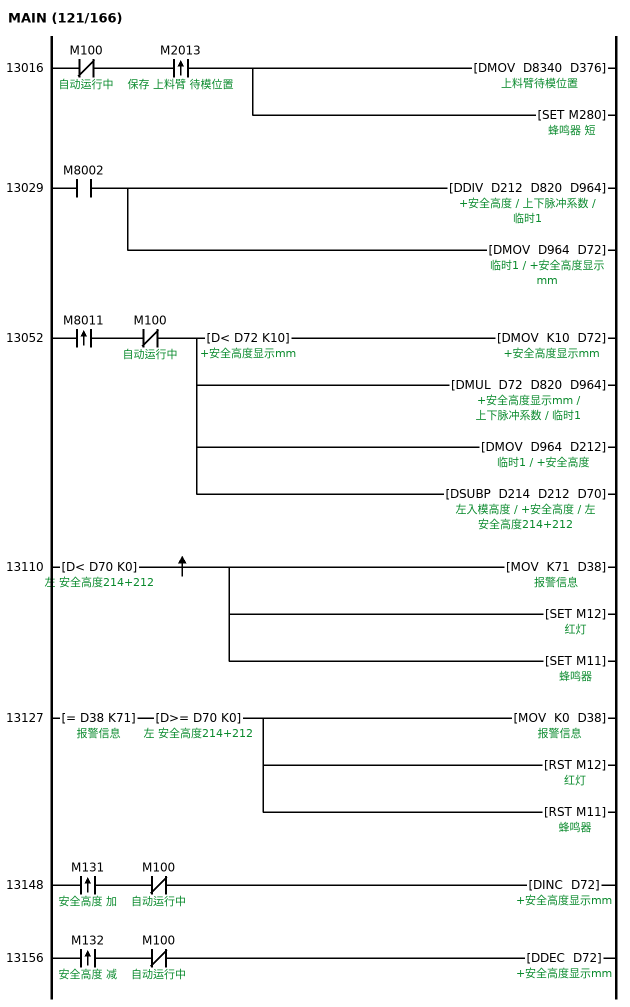
[picture p120: ladder of MAIN, rungs at steps 13016 to 13156]
13016 LDI     M100  ; 自动运行中
      ANDP    M2013  ; 保存 上料臂 待模位置
      DMOV    D8340 D376  ; 上料臂待模位置
      SET     M280  ; 蜂鸣器 短
13029 LD      M8002
      DDIV    D212 D820 D964
      DMOV    D964 D72  ; +安全高度显示mm
13052 LDP     M8011
      ANI     M100  ; 自动运行中
      MPS
      ANDD<   D72 K10  ; +安全高度显示mm
      DMOV    K10 D72
      MPP
      DMUL    D72 D820 D964
      DMOV    D964 D212
      DSUBP   D214 D212 D70
13110 LDD<    D70 K0  ; 左 安全高度214+212
      MEP
      MOV     K71 D38
      SET     M12  ; 红灯
      SET     M11  ; 蜂鸣器
13127 LD=     D38 K71  ; 报警信息
      ANDD>=  D70 K0  ; 左 安全高度214+212
      MOV     K0 D38
      RST     M12  ; 红灯
      RST     M11  ; 蜂鸣器
13148 LDP     M131  ; 安全高度 加
      ANI     M100  ; 自动运行中
      DINC    D72
13156 LDP     M132  ; 安全高度 减
      ANI     M100  ; 自动运行中
      DDEC    D72
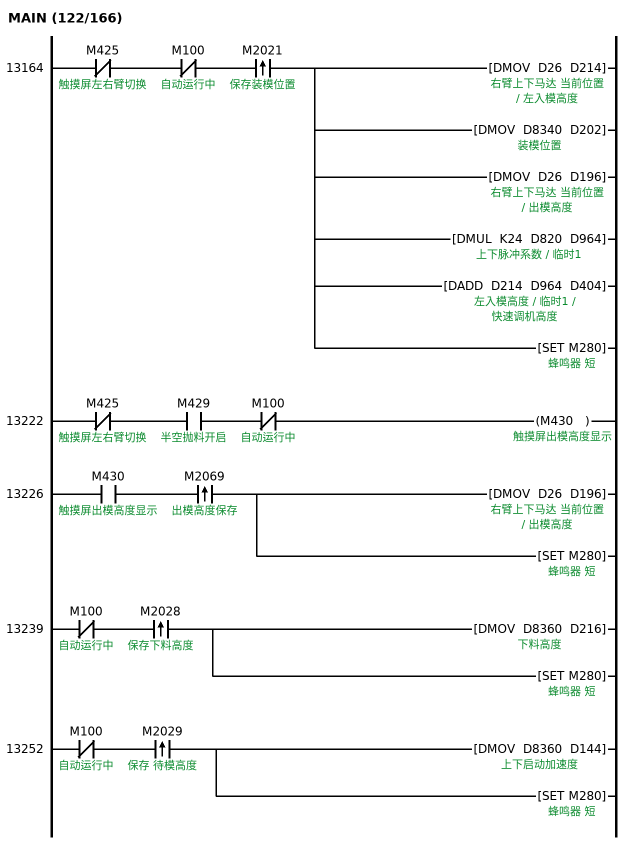
13164 LDI     M425  ; 触摸屏左右臂切换
      ANI     M100  ; 自动运行中
      ANDP    M2021  ; 保存装模位置
      DMOV    D26 D214
      DMOV    D8340 D202
      DMOV    D26 D196
      DMUL    K24 D820 D964
      DADD    D214 D964 D404
      SET     M280  ; 蜂鸣器 短
13222 LDI     M425  ; 触摸屏左右臂切换
      AND     M429  ; 半空抛料开启
      ANI     M100  ; 自动运行中
      OUT     M430  ; 触摸屏出模高度显示
13226 LD      M430  ; 触摸屏出模高度显示
      ANDP    M2069  ; 出模高度保存
      DMOV    D26 D196
      SET     M280  ; 蜂鸣器 短
13239 LDI     M100  ; 自动运行中
      ANDP    M2028  ; 保存下料高度
      DMOV    D8360 D216
      SET     M280  ; 蜂鸣器 短
13252 LDI     M100  ; 自动运行中
      ANDP    M2029  ; 保存 待模高度
      DMOV    D8360 D144  ; 上下启动加速度
      SET     M280  ; 蜂鸣器 短
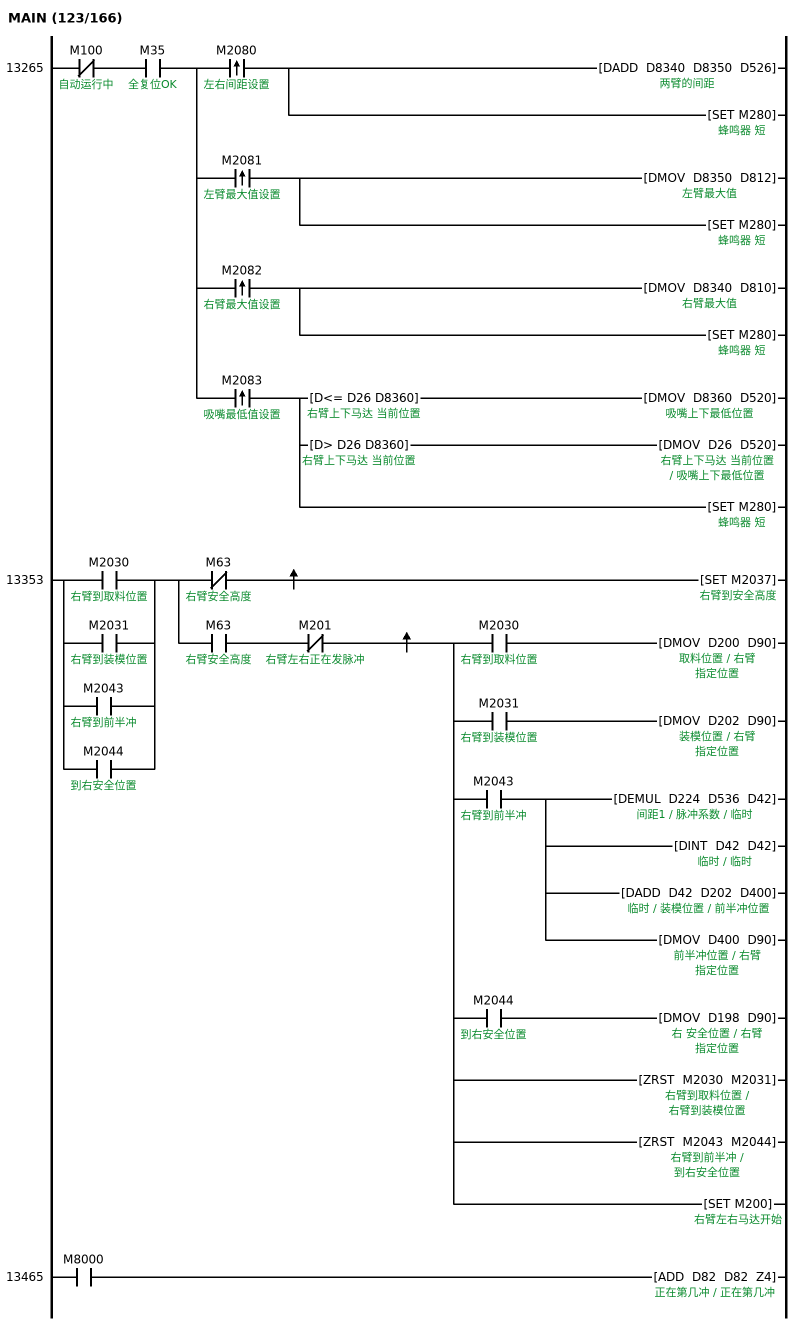
13265 LDI     M100  ; 自动运行中
      AND     M35  ; 全复位OK
      MPS
      ANDP    M2080  ; 左右间距设置
      DADD    D8340 D8350 D526
      SET     M280  ; 蜂鸣器 短
      MRD
      ANDP    M2081  ; 左臂最大值设置
      DMOV    D8350 D812
      SET     M280  ; 蜂鸣器 短
      MRD
      ANDP    M2082  ; 右臂最大值设置
      DMOV    D8340 D810
      SET     M280  ; 蜂鸣器 短
      MPP
      ANDP    M2083  ; 吸嘴最低值设置
      MPS
      ANDD<=  D26 D8360  ; 右臂上下马达 当前位置
      DMOV    D8360 D520
      MRD
      ANDD>   D26 D8360  ; 右臂上下马达 当前位置
      DMOV    D26 D520
      MPP
      SET     M280  ; 蜂鸣器 短
13353 LD      M2030  ; 右臂到取料位置
      OR      M2031  ; 右臂到装模位置
      OR      M2043  ; 右臂到前半冲
      OR      M2044  ; 到右安全位置
      MPS
      ANI     M63  ; 右臂安全高度
      MEP
      SET     M2037  ; 右臂到安全高度
      MPP
      AND     M63  ; 右臂安全高度
      ANI     M201  ; 右臂左右正在发脉冲
      MEP
      MPS
      AND     M2030  ; 右臂到取料位置
      DMOV    D200 D90
      MRD
      AND     M2031  ; 右臂到装模位置
      DMOV    D202 D90
      MRD
      AND     M2043  ; 右臂到前半冲
      DEMUL   D224 D536 D42
      DINT    D42 D42
      DADD    D42 D202 D400
      DMOV    D400 D90
      MRD
      AND     M2044  ; 到右安全位置
      DMOV    D198 D90
      MPP
      ZRST    M2030 M2031
      ZRST    M2043 M2044
      SET     M200  ; 右臂左右马达开始
13465 LD      M8000
      ADD     D82 D82 Z4
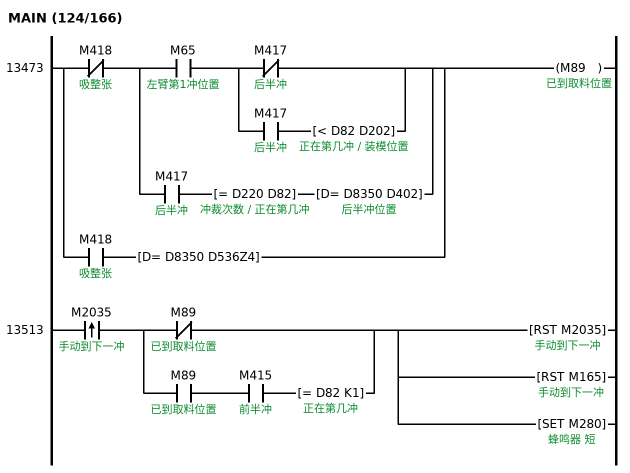
13473 LDI     M418  ; 吸整张
      LD      M65  ; 左臂第1冲位置
      LDI     M417  ; 后半冲
      LD      M417  ; 后半冲
      AND<    D82 D202  ; 正在第几冲 / 装模位置
      ORB
      ANB
      LD      M417  ; 后半冲
      AND=    D220 D82  ; 冲裁次数 / 正在第几冲
      ANDD=   D8350 D402  ; 后半冲位置
      ORB
      ANB
      LD      M418  ; 吸整张
      ANDD=   D8350 D536Z4
      ORB
      OUT     M89  ; 已到取料位置
13513 LDP     M2035  ; 手动到下一冲
      LDI     M89  ; 已到取料位置
      LD      M89  ; 已到取料位置
      AND     M415  ; 前半冲
      AND=    D82 K1  ; 正在第几冲
      ORB
      ANB
      RST     M2035  ; 手动到下一冲
      RST     M165  ; 手动到下一冲
      SET     M280  ; 蜂鸣器 短
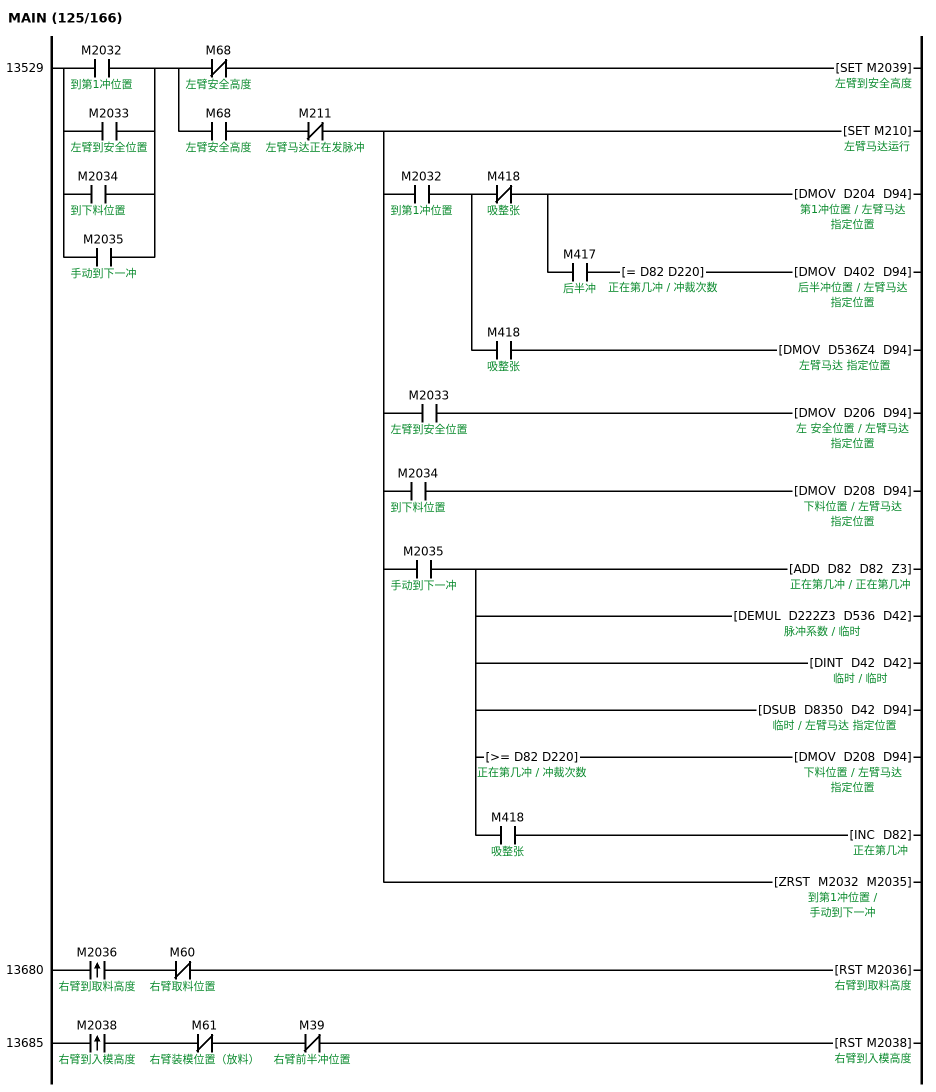
13529 LD      M2032  ; 到第1冲位置
      OR      M2033  ; 左臂到安全位置
      OR      M2034  ; 到下料位置
      OR      M2035  ; 手动到下一冲
      MPS
      ANI     M68  ; 左臂安全高度
      SET     M2039  ; 左臂到安全高度
      MPP
      AND     M68  ; 左臂安全高度
      ANI     M211  ; 左臂马达正在发脉冲
      SET     M210  ; 左臂马达运行
      MPS
      AND     M2032  ; 到第1冲位置
      MPS
      ANI     M418  ; 吸整张
      DMOV    D204 D94
      AND     M417  ; 后半冲
      AND=    D82 D220  ; 正在第几冲 / 冲裁次数
      DMOV    D402 D94
      MPP
      AND     M418  ; 吸整张
      DMOV    D536Z4 D94
      MRD
      AND     M2033  ; 左臂到安全位置
      DMOV    D206 D94
      MRD
      AND     M2034  ; 到下料位置
      DMOV    D208 D94
      MRD
      AND     M2035  ; 手动到下一冲
      ADD     D82 D82 Z3
      DEMUL   D222Z3 D536 D42
      DINT    D42 D42
      DSUB    D8350 D42 D94
      MPS
      AND>=   D82 D220  ; 正在第几冲 / 冲裁次数
      DMOV    D208 D94
      MPP
      AND     M418  ; 吸整张
      INC     D82
      MPP
      ZRST    M2032 M2035
13680 LDP     M2036  ; 右臂到取料高度
      ANI     M60  ; 右臂取料位置
      RST     M2036  ; 右臂到取料高度
13685 LDP     M2038  ; 右臂到入模高度
      ANI     M61  ; 右臂装模位置（放料）
      ANI     M39  ; 右臂前半冲位置
      RST     M2038  ; 右臂到入模高度
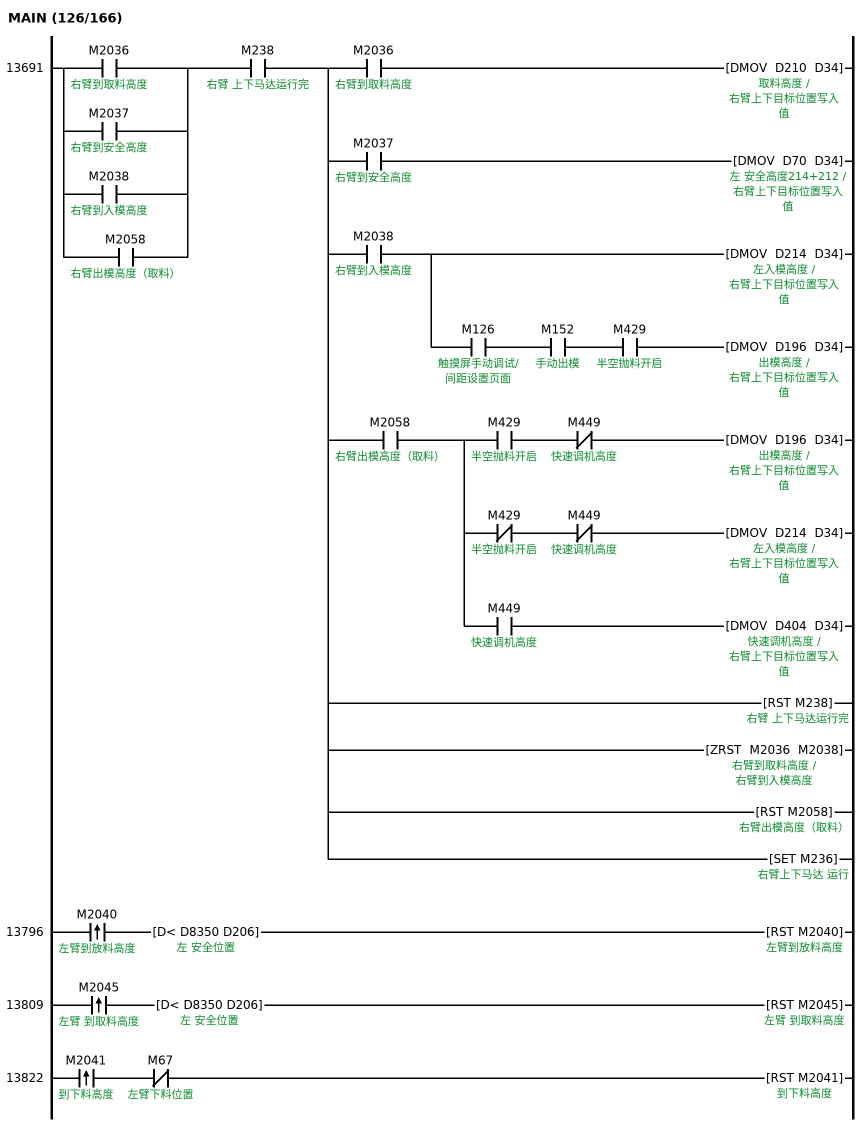
13691 LD      M2036  ; 右臂到取料高度
      OR      M2037  ; 右臂到安全高度
      OR      M2038  ; 右臂到入模高度
      OR      M2058  ; 右臂出模高度（取料）
      AND     M238  ; 右臂 上下马达运行完
      MPS
      AND     M2036  ; 右臂到取料高度
      DMOV    D210 D34
      MRD
      AND     M2037  ; 右臂到安全高度
      DMOV    D70 D34
      MRD
      AND     M2038  ; 右臂到入模高度
      DMOV    D214 D34
      AND     M126  ; 触摸屏手动调试/间距设置页面
      AND     M152  ; 手动出模
      AND     M429  ; 半空抛料开启
      DMOV    D196 D34
      MRD
      AND     M2058  ; 右臂出模高度（取料）
      MPS
      AND     M429  ; 半空抛料开启
      ANI     M449  ; 快速调机高度
      DMOV    D196 D34
      MRD
      ANI     M429  ; 半空抛料开启
      ANI     M449  ; 快速调机高度
      DMOV    D214 D34
      MPP
      AND     M449  ; 快速调机高度
      DMOV    D404 D34
      MPP
      RST     M238  ; 右臂 上下马达运行完
      ZRST    M2036 M2038
      RST     M2058  ; 右臂出模高度（取料）
      SET     M236  ; 右臂上下马达 运行
13796 LDP     M2040  ; 左臂到放料高度
      ANDD<   D8350 D206  ; 左 安全位置
      RST     M2040  ; 左臂到放料高度
13809 LDP     M2045  ; 左臂 到取料高度
      ANDD<   D8350 D206  ; 左 安全位置
      RST     M2045  ; 左臂 到取料高度
13822 LDP     M2041  ; 到下料高度
      ANI     M67  ; 左臂下料位置
      RST     M2041  ; 到下料高度
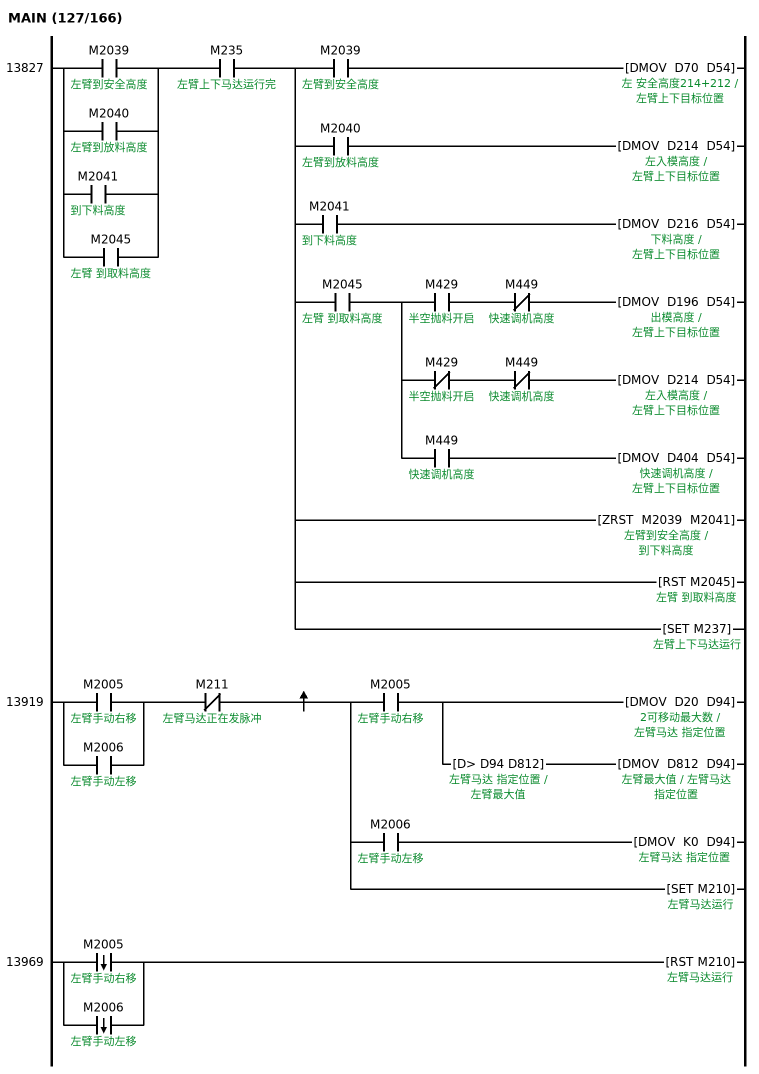
13827 LD      M2039  ; 左臂到安全高度
      OR      M2040  ; 左臂到放料高度
      OR      M2041  ; 到下料高度
      OR      M2045  ; 左臂 到取料高度
      AND     M235  ; 左臂上下马达运行完
      MPS
      AND     M2039  ; 左臂到安全高度
      DMOV    D70 D54
      MRD
      AND     M2040  ; 左臂到放料高度
      DMOV    D214 D54
      MRD
      AND     M2041  ; 到下料高度
      DMOV    D216 D54
      MRD
      AND     M2045  ; 左臂 到取料高度
      MPS
      AND     M429  ; 半空抛料开启
      ANI     M449  ; 快速调机高度
      DMOV    D196 D54
      MRD
      ANI     M429  ; 半空抛料开启
      ANI     M449  ; 快速调机高度
      DMOV    D214 D54
      MPP
      AND     M449  ; 快速调机高度
      DMOV    D404 D54
      MPP
      ZRST    M2039 M2041
      RST     M2045  ; 左臂 到取料高度
      SET     M237  ; 左臂上下马达运行
13919 LD      M2005  ; 左臂手动右移
      OR      M2006  ; 左臂手动左移
      ANI     M211  ; 左臂马达正在发脉冲
      MEP
      MPS
      AND     M2005  ; 左臂手动右移
      DMOV    D20 D94
      ANDD>   D94 D812  ; 左臂马达 指定位置 / 左臂最大值
      DMOV    D812 D94
      MRD
      AND     M2006  ; 左臂手动左移
      DMOV    K0 D94
      MPP
      SET     M210  ; 左臂马达运行
13969 LDF     M2005  ; 左臂手动右移
      ORF     M2006  ; 左臂手动左移
      RST     M210  ; 左臂马达运行
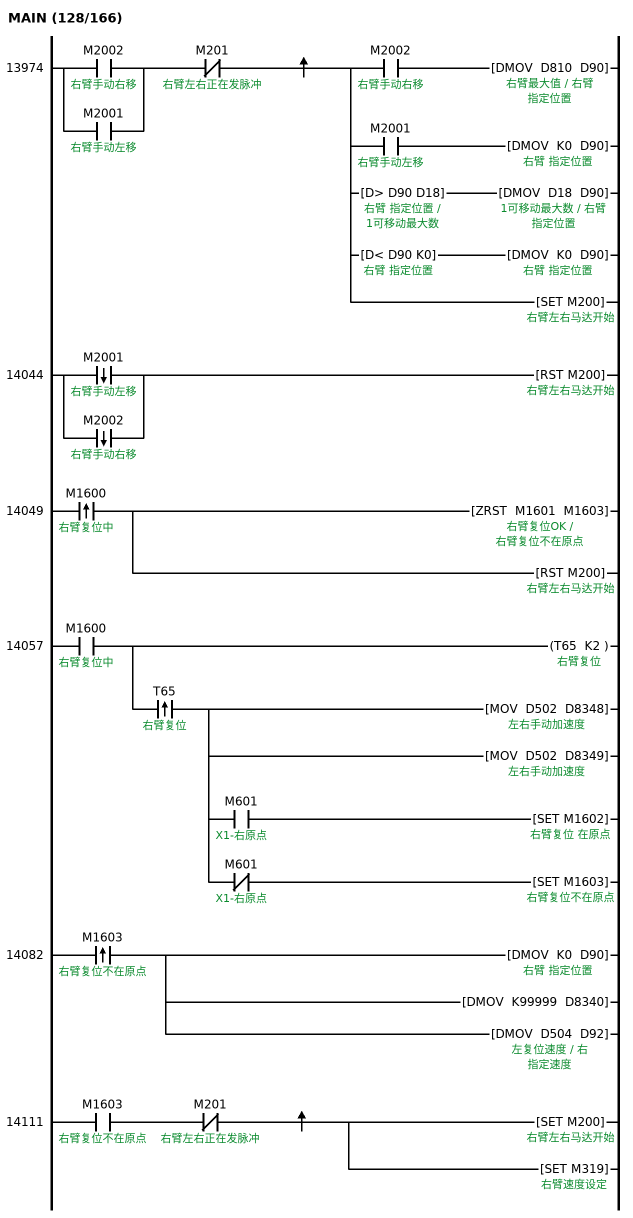
13974 LD      M2002  ; 右臂手动右移
      OR      M2001  ; 右臂手动左移
      ANI     M201  ; 右臂左右正在发脉冲
      MEP
      MPS
      AND     M2002  ; 右臂手动右移
      DMOV    D810 D90
      MRD
      AND     M2001  ; 右臂手动左移
      DMOV    K0 D90
      MRD
      ANDD>   D90 D18  ; 右臂 指定位置 / 1可移动最大数
      DMOV    D18 D90
      MRD
      ANDD<   D90 K0  ; 右臂 指定位置
      DMOV    K0 D90
      MPP
      SET     M200  ; 右臂左右马达开始
14044 LDF     M2001  ; 右臂手动左移
      ORF     M2002  ; 右臂手动右移
      RST     M200  ; 右臂左右马达开始
14049 LDP     M1600  ; 右臂复位中
      ZRST    M1601 M1603  ; 右臂复位不在原点
      RST     M200  ; 右臂左右马达开始
14057 LD      M1600  ; 右臂复位中
      OUT     T65 K2  ; 右臂复位
      ANDP    T65  ; 右臂复位
      MOV     D502 D8348
      MOV     D502 D8349
      MPS
      AND     M601  ; X1-右原点
      SET     M1602  ; 右臂复位 在原点
      MPP
      ANI     M601  ; X1-右原点
      SET     M1603  ; 右臂复位不在原点
14082 LDP     M1603  ; 右臂复位不在原点
      DMOV    K0 D90
      DMOV    K99999 D8340
      DMOV    D504 D92  ; 右 指定速度
14111 LD      M1603  ; 右臂复位不在原点
      ANI     M201  ; 右臂左右正在发脉冲
      MEP
      SET     M200  ; 右臂左右马达开始
      SET     M319  ; 右臂速度设定
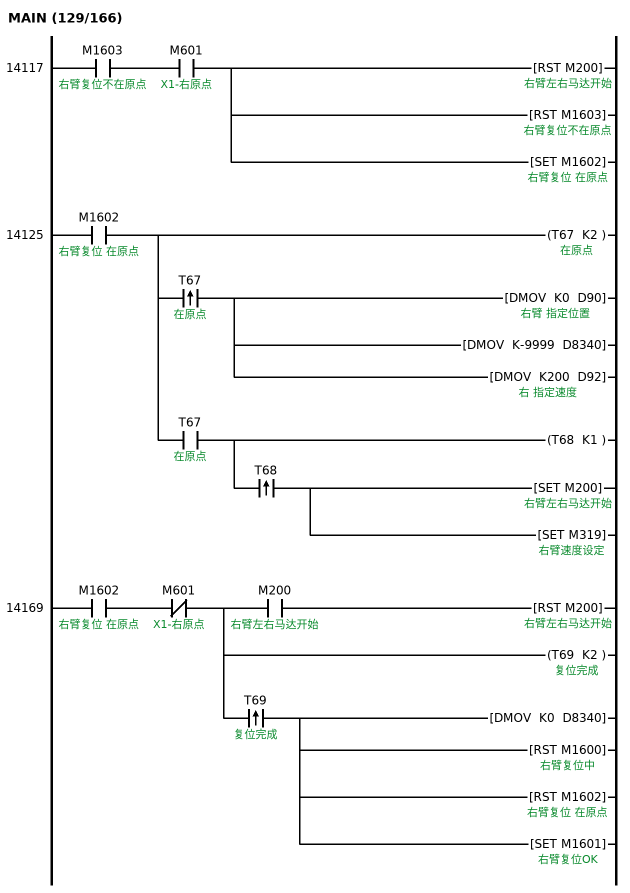
14117 LD      M1603  ; 右臂复位不在原点
      AND     M601  ; X1-右原点
      RST     M200  ; 右臂左右马达开始
      RST     M1603  ; 右臂复位不在原点
      SET     M1602  ; 右臂复位 在原点
14125 LD      M1602  ; 右臂复位 在原点
      OUT     T67 K2  ; 在原点
      MPS
      ANDP    T67  ; 在原点
      DMOV    K0 D90
      DMOV    K-9999 D8340
      DMOV    K200 D92
      MPP
      AND     T67  ; 在原点
      OUT     T68 K1
      ANDP    T68
      SET     M200  ; 右臂左右马达开始
      SET     M319  ; 右臂速度设定
14169 LD      M1602  ; 右臂复位 在原点
      ANI     M601  ; X1-右原点
      MPS
      AND     M200  ; 右臂左右马达开始
      RST     M200  ; 右臂左右马达开始
      MPP
      OUT     T69 K2  ; 复位完成
      ANDP    T69  ; 复位完成
      DMOV    K0 D8340
      RST     M1600  ; 右臂复位中
      RST     M1602  ; 右臂复位 在原点
      SET     M1601  ; 右臂复位OK
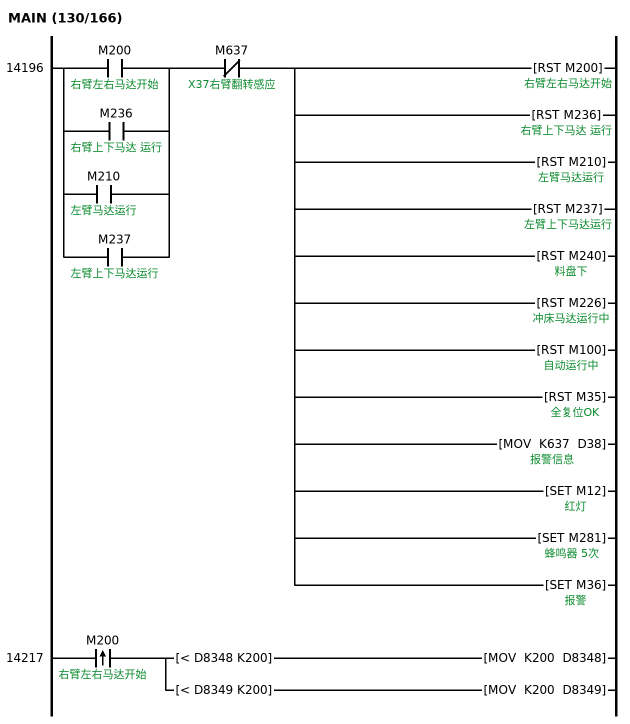
14196 LD      M200  ; 右臂左右马达开始
      OR      M236  ; 右臂上下马达 运行
      OR      M210  ; 左臂马达运行
      OR      M237  ; 左臂上下马达运行
      ANI     M637  ; X37右臂翻转感应
      RST     M200  ; 右臂左右马达开始
      RST     M236  ; 右臂上下马达 运行
      RST     M210  ; 左臂马达运行
      RST     M237  ; 左臂上下马达运行
      RST     M240  ; 料盘下
      RST     M226  ; 冲床马达运行中
      RST     M100  ; 自动运行中
      RST     M35  ; 全复位OK
      MOV     K637 D38
      SET     M12  ; 红灯
      SET     M281  ; 蜂鸣器 5次
      SET     M36  ; 报警
14217 LDP     M200  ; 右臂左右马达开始
      MPS
      AND<    D8348 K200
      MOV     K200 D8348
      MPP
      AND<    D8349 K200
      MOV     K200 D8349
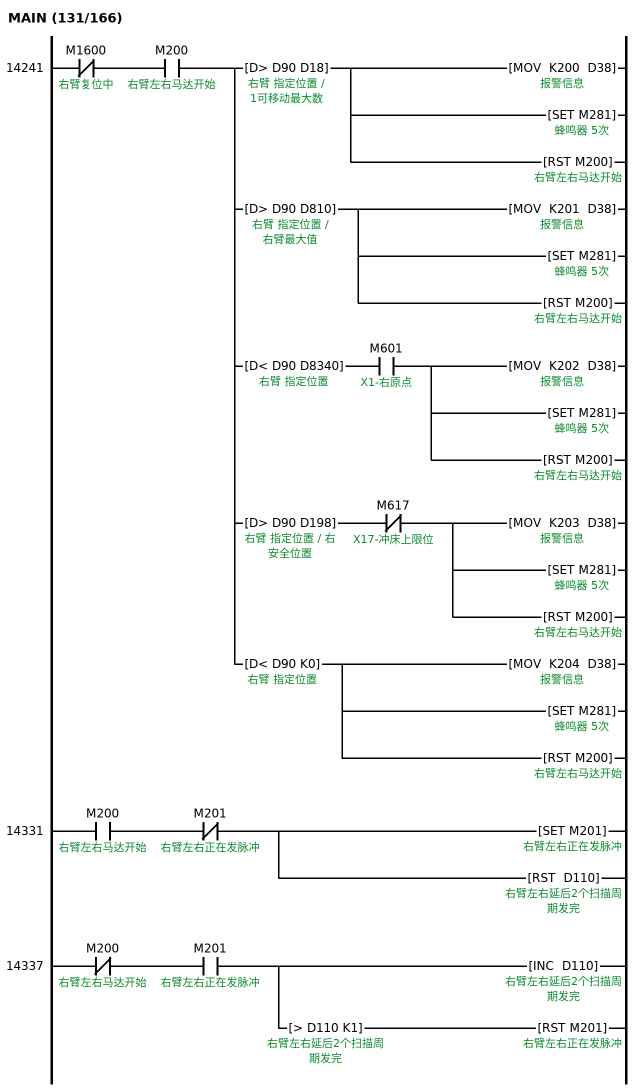
14241 LDI     M1600  ; 右臂复位中
      AND     M200  ; 右臂左右马达开始
      MPS
      ANDD>   D90 D18  ; 右臂 指定位置 / 1可移动最大数
      MOV     K200 D38
      SET     M281  ; 蜂鸣器 5次
      RST     M200  ; 右臂左右马达开始
      MRD
      ANDD>   D90 D810  ; 右臂 指定位置 / 右臂最大值
      MOV     K201 D38
      SET     M281  ; 蜂鸣器 5次
      RST     M200  ; 右臂左右马达开始
      MRD
      ANDD<   D90 D8340  ; 右臂 指定位置
      AND     M601  ; X1-右原点
      MOV     K202 D38
      SET     M281  ; 蜂鸣器 5次
      RST     M200  ; 右臂左右马达开始
      MRD
      ANDD>   D90 D198  ; 右臂 指定位置 / 右 安全位置
      ANI     M617  ; X17-冲床上限位
      MOV     K203 D38
      SET     M281  ; 蜂鸣器 5次
      RST     M200  ; 右臂左右马达开始
      MPP
      ANDD<   D90 K0  ; 右臂 指定位置
      MOV     K204 D38
      SET     M281  ; 蜂鸣器 5次
      RST     M200  ; 右臂左右马达开始
14331 LD      M200  ; 右臂左右马达开始
      ANI     M201  ; 右臂左右正在发脉冲
      SET     M201  ; 右臂左右正在发脉冲
      RST     D110  ; 右臂左右延后2个扫描周期发完
14337 LDI     M200  ; 右臂左右马达开始
      AND     M201  ; 右臂左右正在发脉冲
      INC     D110
      AND>    D110 K1  ; 右臂左右延后2个扫描周期发完
      RST     M201  ; 右臂左右正在发脉冲
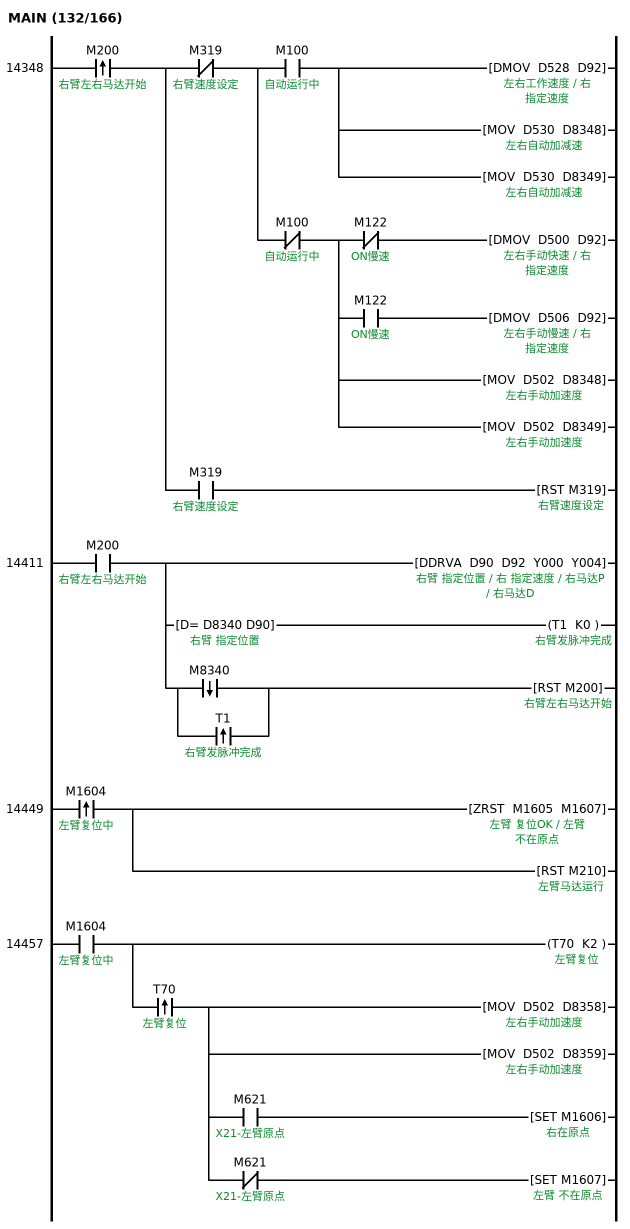
14348 LDP     M200  ; 右臂左右马达开始
      MPS
      ANI     M319  ; 右臂速度设定
      MPS
      AND     M100  ; 自动运行中
      DMOV    D528 D92
      MOV     D530 D8348
      MOV     D530 D8349
      MPP
      ANI     M100  ; 自动运行中
      MPS
      ANI     M122  ; ON慢速
      DMOV    D500 D92
      MRD
      AND     M122  ; ON慢速
      DMOV    D506 D92
      MPP
      MOV     D502 D8348
      MOV     D502 D8349
      MPP
      AND     M319  ; 右臂速度设定
      RST     M319  ; 右臂速度设定
14411 LD      M200  ; 右臂左右马达开始
      DDRVA   D90 D92 Y000 Y004  ; 右马达P / 右马达D
      MPS
      ANDD=   D8340 D90  ; 右臂 指定位置
      OUT     T1 K0  ; 右臂发脉冲完成
      MPP
      LDF     M8340
      ORP     T1  ; 右臂发脉冲完成
      ANB
      RST     M200  ; 右臂左右马达开始
14449 LDP     M1604  ; 左臂复位中
      ZRST    M1605 M1607  ; 左臂 不在原点
      RST     M210  ; 左臂马达运行
14457 LD      M1604  ; 左臂复位中
      OUT     T70 K2  ; 左臂复位
      ANDP    T70  ; 左臂复位
      MOV     D502 D8358
      MOV     D502 D8359
      MPS
      AND     M621  ; X21-左臂原点
      SET     M1606  ; 右在原点
      MPP
      ANI     M621  ; X21-左臂原点
      SET     M1607  ; 左臂 不在原点
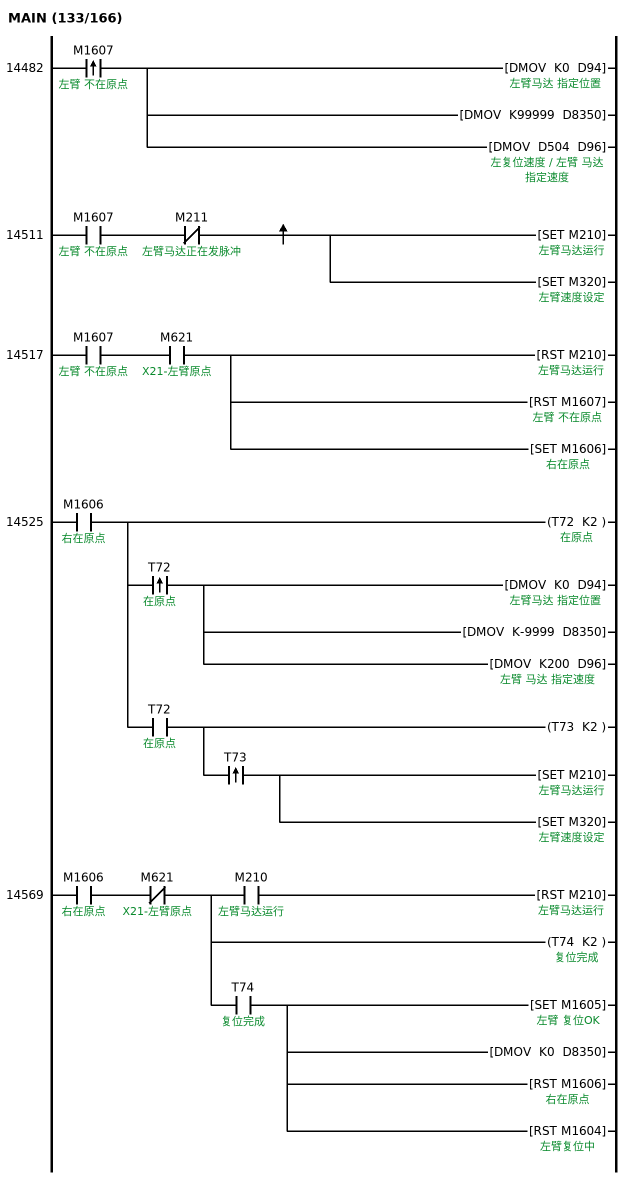
14482 LDP     M1607  ; 左臂 不在原点
      DMOV    K0 D94
      DMOV    K99999 D8350
      DMOV    D504 D96  ; 左臂 马达 指定速度
14511 LD      M1607  ; 左臂 不在原点
      ANI     M211  ; 左臂马达正在发脉冲
      MEP
      SET     M210  ; 左臂马达运行
      SET     M320  ; 左臂速度设定
14517 LD      M1607  ; 左臂 不在原点
      AND     M621  ; X21-左臂原点
      RST     M210  ; 左臂马达运行
      RST     M1607  ; 左臂 不在原点
      SET     M1606  ; 右在原点
14525 LD      M1606  ; 右在原点
      OUT     T72 K2  ; 在原点
      MPS
      ANDP    T72  ; 在原点
      DMOV    K0 D94
      DMOV    K-9999 D8350
      DMOV    K200 D96
      MPP
      AND     T72  ; 在原点
      OUT     T73 K2
      ANDP    T73
      SET     M210  ; 左臂马达运行
      SET     M320  ; 左臂速度设定
14569 LD      M1606  ; 右在原点
      ANI     M621  ; X21-左臂原点
      MPS
      AND     M210  ; 左臂马达运行
      RST     M210  ; 左臂马达运行
      MPP
      OUT     T74 K2  ; 复位完成
      AND     T74  ; 复位完成
      SET     M1605  ; 左臂 复位OK
      DMOV    K0 D8350
      RST     M1606  ; 右在原点
      RST     M1604  ; 左臂复位中
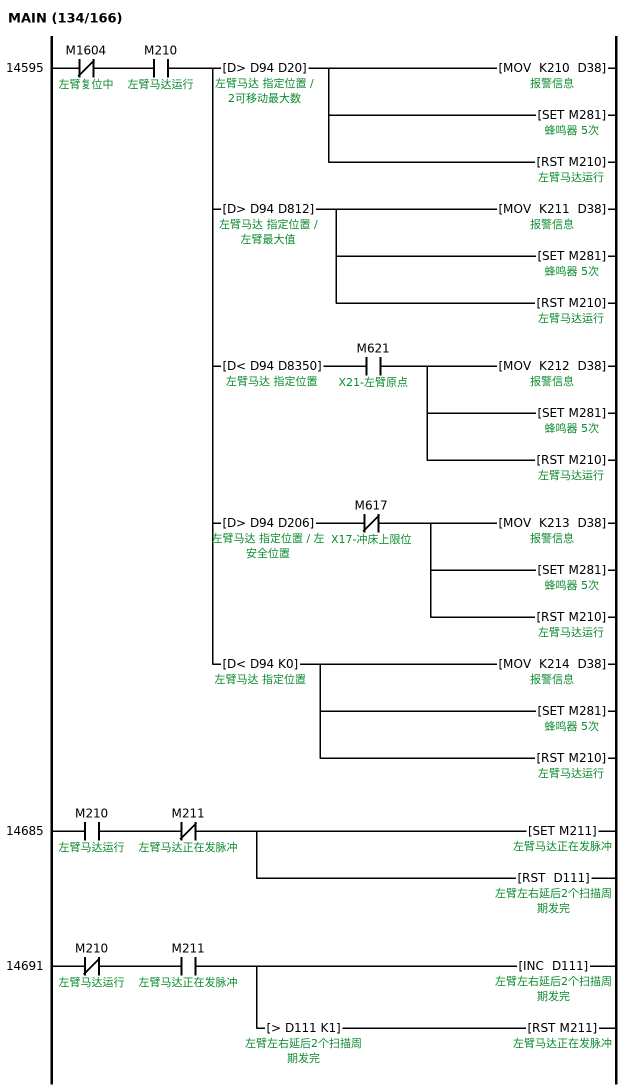
14595 LDI     M1604  ; 左臂复位中
      AND     M210  ; 左臂马达运行
      MPS
      ANDD>   D94 D20  ; 左臂马达 指定位置 / 2可移动最大数
      MOV     K210 D38
      SET     M281  ; 蜂鸣器 5次
      RST     M210  ; 左臂马达运行
      MRD
      ANDD>   D94 D812  ; 左臂马达 指定位置 / 左臂最大值
      MOV     K211 D38
      SET     M281  ; 蜂鸣器 5次
      RST     M210  ; 左臂马达运行
      MRD
      ANDD<   D94 D8350  ; 左臂马达 指定位置
      AND     M621  ; X21-左臂原点
      MOV     K212 D38
      SET     M281  ; 蜂鸣器 5次
      RST     M210  ; 左臂马达运行
      MRD
      ANDD>   D94 D206  ; 左臂马达 指定位置 / 左 安全位置
      ANI     M617  ; X17-冲床上限位
      MOV     K213 D38
      SET     M281  ; 蜂鸣器 5次
      RST     M210  ; 左臂马达运行
      MPP
      ANDD<   D94 K0  ; 左臂马达 指定位置
      MOV     K214 D38
      SET     M281  ; 蜂鸣器 5次
      RST     M210  ; 左臂马达运行
14685 LD      M210  ; 左臂马达运行
      ANI     M211  ; 左臂马达正在发脉冲
      SET     M211  ; 左臂马达正在发脉冲
      RST     D111  ; 左臂左右延后2个扫描周期发完
14691 LDI     M210  ; 左臂马达运行
      AND     M211  ; 左臂马达正在发脉冲
      INC     D111
      AND>    D111 K1  ; 左臂左右延后2个扫描周期发完
      RST     M211  ; 左臂马达正在发脉冲
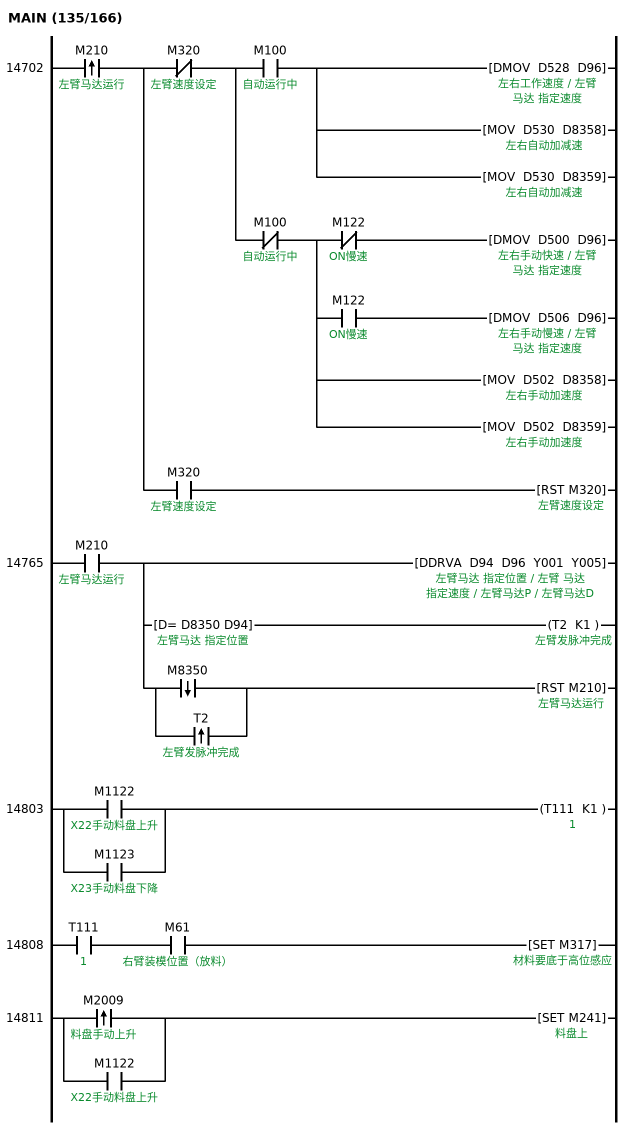
14702 LDP     M210  ; 左臂马达运行
      MPS
      ANI     M320  ; 左臂速度设定
      MPS
      AND     M100  ; 自动运行中
      DMOV    D528 D96
      MOV     D530 D8358
      MOV     D530 D8359
      MPP
      ANI     M100  ; 自动运行中
      MPS
      ANI     M122  ; ON慢速
      DMOV    D500 D96
      MRD
      AND     M122  ; ON慢速
      DMOV    D506 D96
      MPP
      MOV     D502 D8358
      MOV     D502 D8359
      MPP
      AND     M320  ; 左臂速度设定
      RST     M320  ; 左臂速度设定
14765 LD      M210  ; 左臂马达运行
      DDRVA   D94 D96 Y001 Y005  ; 左臂马达P / 左臂马达D
      MPS
      ANDD=   D8350 D94  ; 左臂马达 指定位置
      OUT     T2 K1  ; 左臂发脉冲完成
      MPP
      LDF     M8350
      ORP     T2  ; 左臂发脉冲完成
      ANB
      RST     M210  ; 左臂马达运行
14803 LD      M1122  ; X22手动料盘上升
      OR      M1123  ; X23手动料盘下降
      OUT     T111 K1  ; 1
14808 LD      T111  ; 1
      AND     M61  ; 右臂装模位置（放料）
      SET     M317  ; 材料要底于高位感应
14811 LDP     M2009  ; 料盘手动上升
      OR      M1122  ; X22手动料盘上升
      SET     M241  ; 料盘上
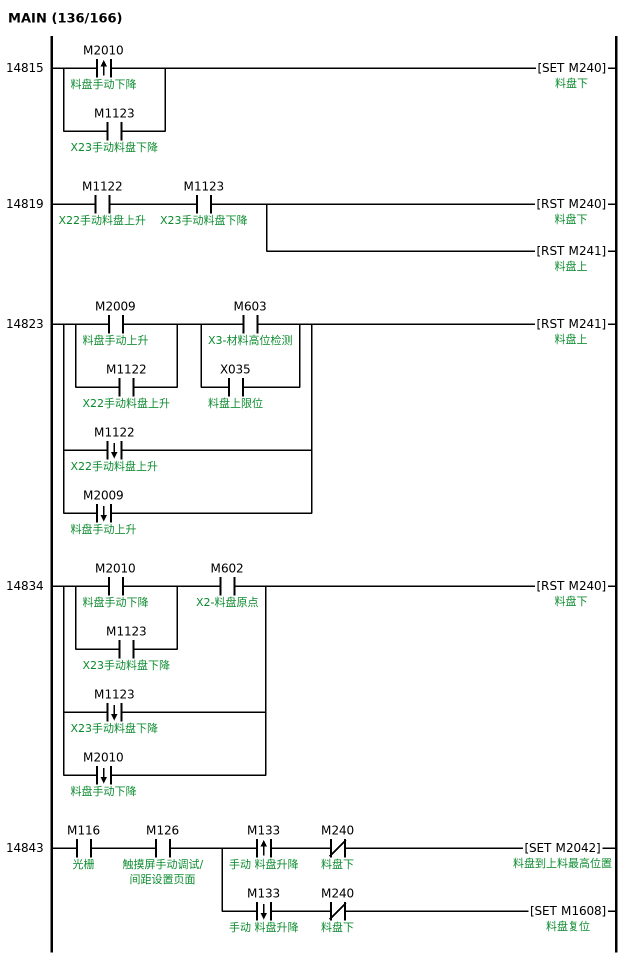
14815 LDP     M2010  ; 料盘手动下降
      OR      M1123  ; X23手动料盘下降
      SET     M240  ; 料盘下
14819 LD      M1122  ; X22手动料盘上升
      AND     M1123  ; X23手动料盘下降
      RST     M240  ; 料盘下
      RST     M241  ; 料盘上
14823 LD      M2009  ; 料盘手动上升
      OR      M1122  ; X22手动料盘上升
      LD      M603  ; X3-材料高位检测
      OR      X035  ; 料盘上限位
      ANB
      ORF     M1122  ; X22手动料盘上升
      ORF     M2009  ; 料盘手动上升
      RST     M241  ; 料盘上
14834 LD      M2010  ; 料盘手动下降
      OR      M1123  ; X23手动料盘下降
      AND     M602  ; X2-料盘原点
      ORF     M1123  ; X23手动料盘下降
      ORF     M2010  ; 料盘手动下降
      RST     M240  ; 料盘下
14843 LD      M116  ; 光栅
      AND     M126  ; 触摸屏手动调试/间距设置页面
      MPS
      ANDP    M133  ; 手动 料盘升降
      ANI     M240  ; 料盘下
      SET     M2042  ; 料盘到上料最高位置
      MPP
      ANDF    M133  ; 手动 料盘升降
      ANI     M240  ; 料盘下
      SET     M1608  ; 料盘复位
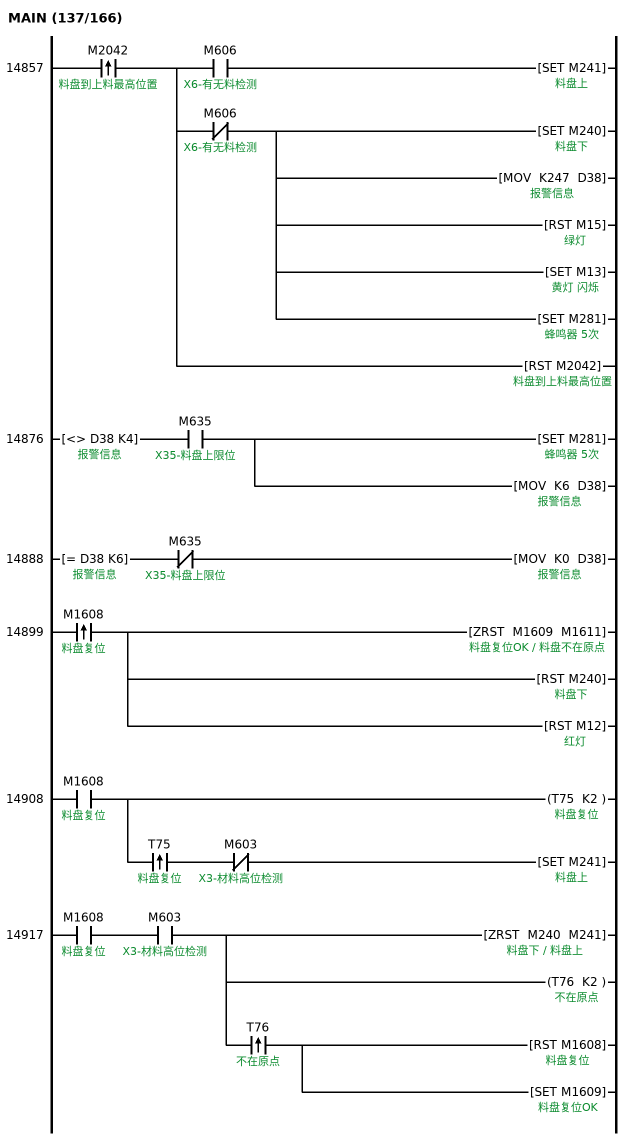
14857 LDP     M2042  ; 料盘到上料最高位置
      MPS
      AND     M606  ; X6-有无料检测
      SET     M241  ; 料盘上
      MRD
      ANI     M606  ; X6-有无料检测
      SET     M240  ; 料盘下
      MOV     K247 D38
      RST     M15  ; 绿灯
      SET     M13  ; 黄灯 闪烁
      SET     M281  ; 蜂鸣器 5次
      MPP
      RST     M2042  ; 料盘到上料最高位置
14876 LD<>    D38 K4  ; 报警信息
      AND     M635  ; X35-料盘上限位
      SET     M281  ; 蜂鸣器 5次
      MOV     K6 D38
14888 LD=     D38 K6  ; 报警信息
      ANI     M635  ; X35-料盘上限位
      MOV     K0 D38
14899 LDP     M1608  ; 料盘复位
      ZRST    M1609 M1611
      RST     M240  ; 料盘下
      RST     M12  ; 红灯
14908 LD      M1608  ; 料盘复位
      OUT     T75 K2  ; 料盘复位
      ANDP    T75  ; 料盘复位
      ANI     M603  ; X3-材料高位检测
      SET     M241  ; 料盘上
14917 LD      M1608  ; 料盘复位
      AND     M603  ; X3-材料高位检测
      ZRST    M240 M241
      OUT     T76 K2  ; 不在原点
      ANDP    T76  ; 不在原点
      RST     M1608  ; 料盘复位
      SET     M1609  ; 料盘复位OK
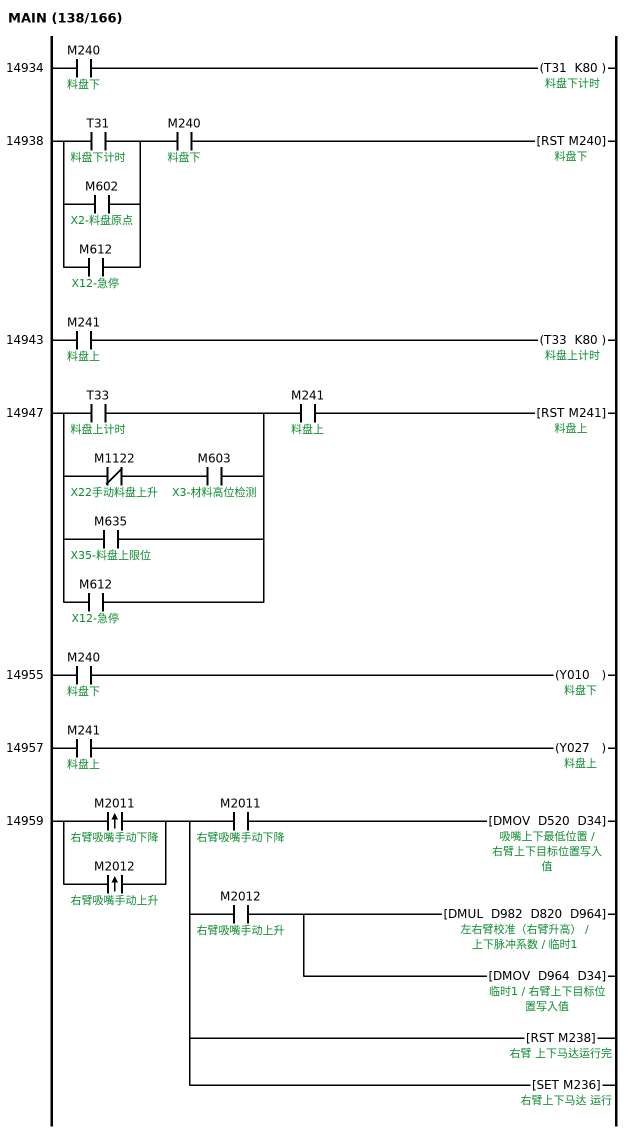
14934 LD      M240  ; 料盘下
      OUT     T31 K80  ; 料盘下计时
14938 LD      T31  ; 料盘下计时
      OR      M602  ; X2-料盘原点
      OR      M612  ; X12-急停
      AND     M240  ; 料盘下
      RST     M240  ; 料盘下
14943 LD      M241  ; 料盘上
      OUT     T33 K80  ; 料盘上计时
14947 LD      T33  ; 料盘上计时
      LDI     M1122  ; X22手动料盘上升
      AND     M603  ; X3-材料高位检测
      ORB
      OR      M635  ; X35-料盘上限位
      OR      M612  ; X12-急停
      AND     M241  ; 料盘上
      RST     M241  ; 料盘上
14955 LD      M240  ; 料盘下
      OUT     Y010  ; 料盘下
14957 LD      M241  ; 料盘上
      OUT     Y027  ; 料盘上
14959 LDP     M2011  ; 右臂吸嘴手动下降
      ORP     M2012  ; 右臂吸嘴手动上升
      MPS
      AND     M2011  ; 右臂吸嘴手动下降
      DMOV    D520 D34
      MRD
      AND     M2012  ; 右臂吸嘴手动上升
      DMUL    D982 D820 D964  ; 左右臂校准（右臂升高）
      DMOV    D964 D34
      MPP
      RST     M238  ; 右臂 上下马达运行完
      SET     M236  ; 右臂上下马达 运行
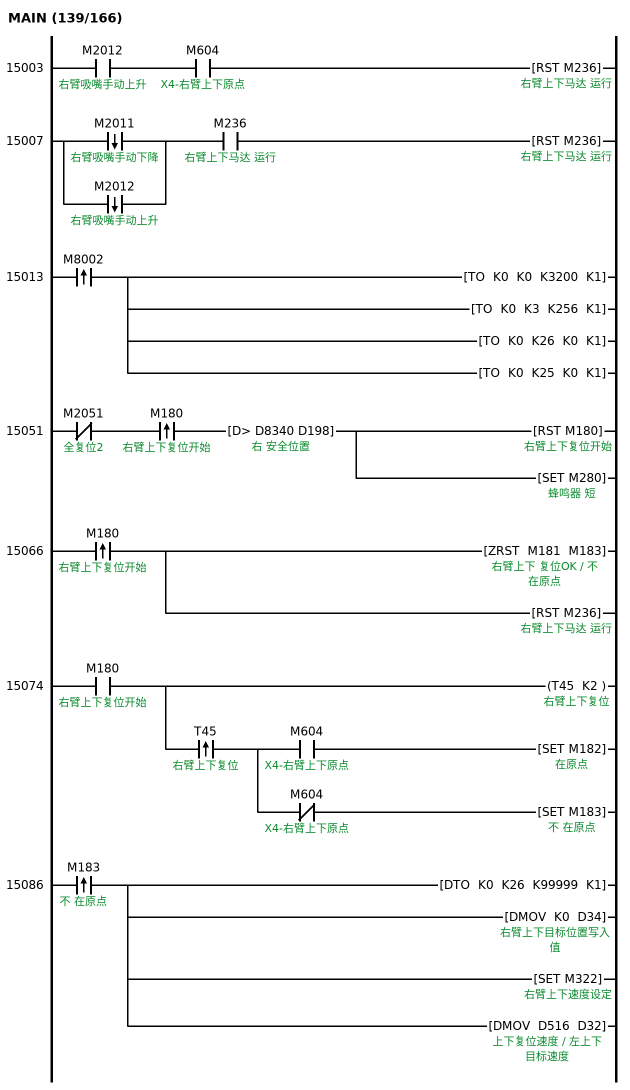
15003 LD      M2012  ; 右臂吸嘴手动上升
      AND     M604  ; X4-右臂上下原点
      RST     M236  ; 右臂上下马达 运行
15007 LDF     M2011  ; 右臂吸嘴手动下降
      ORF     M2012  ; 右臂吸嘴手动上升
      AND     M236  ; 右臂上下马达 运行
      RST     M236  ; 右臂上下马达 运行
15013 LDP     M8002
      TO      K0 K0 K3200 K1
      TO      K0 K3 K256 K1
      TO      K0 K26 K0 K1
      TO      K0 K25 K0 K1
15051 LDI     M2051  ; 全复位2
      ANDP    M180  ; 右臂上下复位开始
      ANDD>   D8340 D198  ; 右 安全位置
      RST     M180  ; 右臂上下复位开始
      SET     M280  ; 蜂鸣器 短
15066 LDP     M180  ; 右臂上下复位开始
      ZRST    M181 M183  ; 不 在原点
      RST     M236  ; 右臂上下马达 运行
15074 LD      M180  ; 右臂上下复位开始
      OUT     T45 K2  ; 右臂上下复位
      ANDP    T45  ; 右臂上下复位
      MPS
      AND     M604  ; X4-右臂上下原点
      SET     M182  ; 在原点
      MPP
      ANI     M604  ; X4-右臂上下原点
      SET     M183  ; 不 在原点
15086 LDP     M183  ; 不 在原点
      DTO     K0 K26 K99999 K1
      DMOV    K0 D34
      SET     M322  ; 右臂上下速度设定
      DMOV    D516 D32
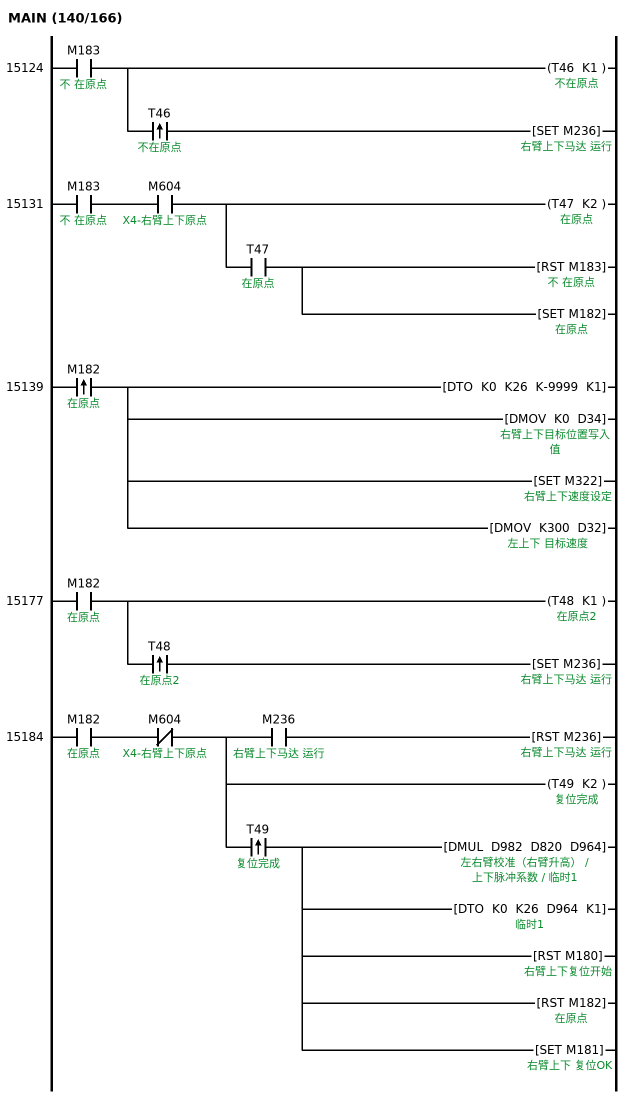
15124 LD      M183  ; 不 在原点
      OUT     T46 K1  ; 不在原点
      ANDP    T46  ; 不在原点
      SET     M236  ; 右臂上下马达 运行
15131 LD      M183  ; 不 在原点
      AND     M604  ; X4-右臂上下原点
      OUT     T47 K2  ; 在原点
      AND     T47  ; 在原点
      RST     M183  ; 不 在原点
      SET     M182  ; 在原点
15139 LDP     M182  ; 在原点
      DTO     K0 K26 K-9999 K1
      DMOV    K0 D34
      SET     M322  ; 右臂上下速度设定
      DMOV    K300 D32
15177 LD      M182  ; 在原点
      OUT     T48 K1  ; 在原点2
      ANDP    T48  ; 在原点2
      SET     M236  ; 右臂上下马达 运行
15184 LD      M182  ; 在原点
      ANI     M604  ; X4-右臂上下原点
      MPS
      AND     M236  ; 右臂上下马达 运行
      RST     M236  ; 右臂上下马达 运行
      MPP
      OUT     T49 K2  ; 复位完成
      ANDP    T49  ; 复位完成
      DMUL    D982 D820 D964
      DTO     K0 K26 D964 K1
      RST     M180  ; 右臂上下复位开始
      RST     M182  ; 在原点
      SET     M181  ; 右臂上下 复位OK
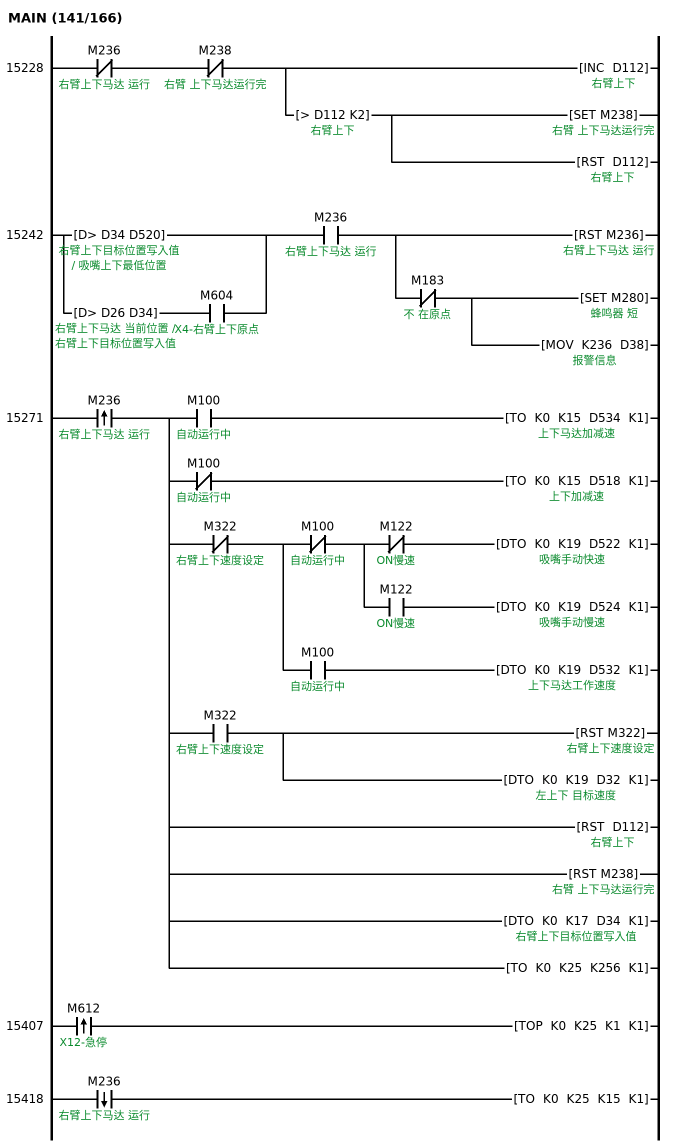
15228 LDI     M236  ; 右臂上下马达 运行
      ANI     M238  ; 右臂 上下马达运行完
      INC     D112  ; 右臂上下
      AND>    D112 K2  ; 右臂上下
      SET     M238  ; 右臂 上下马达运行完
      RST     D112  ; 右臂上下
15242 LDD>    D34 D520  ; 右臂上下目标位置写入值 / 吸嘴上下最低位置
      LDD>    D26 D34  ; 右臂上下马达 当前位置 / 右臂上下目标位置写入值
      AND     M604  ; X4-右臂上下原点
      ORB
      AND     M236  ; 右臂上下马达 运行
      RST     M236  ; 右臂上下马达 运行
      ANI     M183  ; 不 在原点
      SET     M280  ; 蜂鸣器 短
      MOV     K236 D38
15271 LDP     M236  ; 右臂上下马达 运行
      MPS
      AND     M100  ; 自动运行中
      TO      K0 K15 D534 K1
      MRD
      ANI     M100  ; 自动运行中
      TO      K0 K15 D518 K1
      MRD
      ANI     M322  ; 右臂上下速度设定
      MPS
      ANI     M100  ; 自动运行中
      MPS
      ANI     M122  ; ON慢速
      DTO     K0 K19 D522 K1
      MPP
      AND     M122  ; ON慢速
      DTO     K0 K19 D524 K1
      MPP
      AND     M100  ; 自动运行中
      DTO     K0 K19 D532 K1
      MRD
      AND     M322  ; 右臂上下速度设定
      RST     M322  ; 右臂上下速度设定
      DTO     K0 K19 D32 K1
      MPP
      RST     D112  ; 右臂上下
      RST     M238  ; 右臂 上下马达运行完
      DTO     K0 K17 D34 K1
      TO      K0 K25 K256 K1
15407 LDP     M612  ; X12-急停
      TOP     K0 K25 K1 K1
15418 LDF     M236  ; 右臂上下马达 运行
      TO      K0 K25 K15 K1
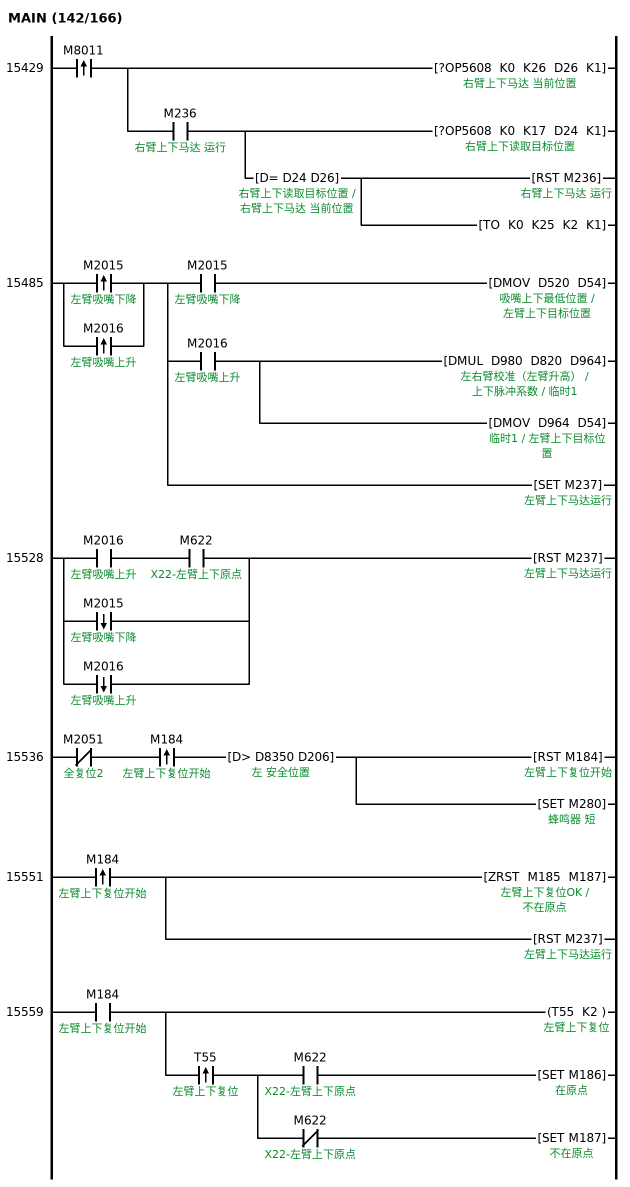
15429 LDP     M8011
      ?OP5608 K0 K26 D26 K1
      AND     M236  ; 右臂上下马达 运行
      ?OP5608 K0 K17 D24 K1  ; 右臂上下读取目标位置
      ANDD=   D24 D26  ; 右臂上下读取目标位置 / 右臂上下马达 当前位置
      RST     M236  ; 右臂上下马达 运行
      TO      K0 K25 K2 K1
15485 LDP     M2015  ; 左臂吸嘴下降
      ORP     M2016  ; 左臂吸嘴上升
      MPS
      AND     M2015  ; 左臂吸嘴下降
      DMOV    D520 D54
      MRD
      AND     M2016  ; 左臂吸嘴上升
      DMUL    D980 D820 D964  ; 左右臂校准（左臂升高）
      DMOV    D964 D54
      MPP
      SET     M237  ; 左臂上下马达运行
15528 LD      M2016  ; 左臂吸嘴上升
      AND     M622  ; X22-左臂上下原点
      ORF     M2015  ; 左臂吸嘴下降
      ORF     M2016  ; 左臂吸嘴上升
      RST     M237  ; 左臂上下马达运行
15536 LDI     M2051  ; 全复位2
      ANDP    M184  ; 左臂上下复位开始
      ANDD>   D8350 D206  ; 左 安全位置
      RST     M184  ; 左臂上下复位开始
      SET     M280  ; 蜂鸣器 短
15551 LDP     M184  ; 左臂上下复位开始
      ZRST    M185 M187
      RST     M237  ; 左臂上下马达运行
15559 LD      M184  ; 左臂上下复位开始
      OUT     T55 K2  ; 左臂上下复位
      ANDP    T55  ; 左臂上下复位
      MPS
      AND     M622  ; X22-左臂上下原点
      SET     M186  ; 在原点
      MPP
      ANI     M622  ; X22-左臂上下原点
      SET     M187  ; 不在原点
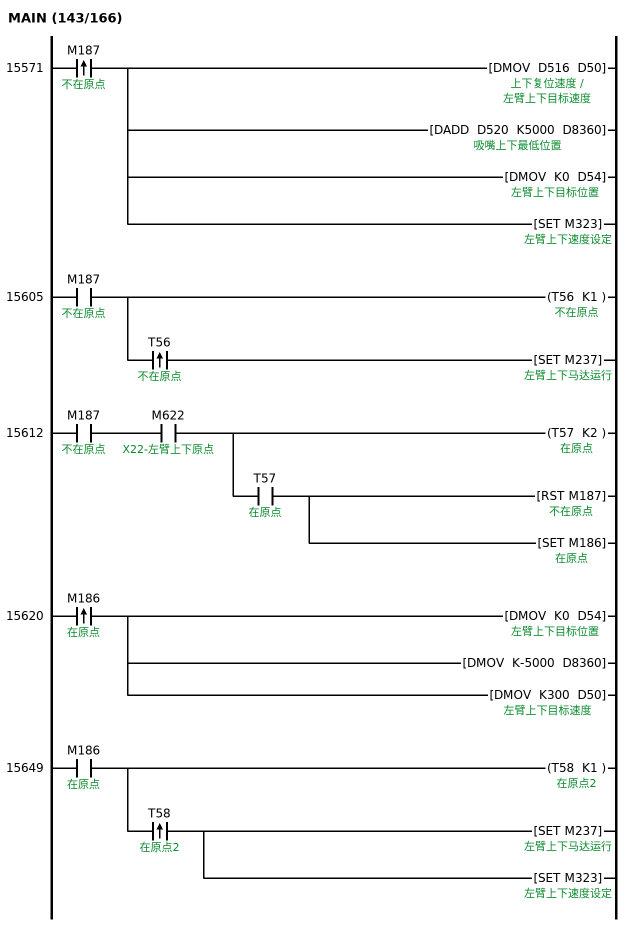
15571 LDP     M187  ; 不在原点
      DMOV    D516 D50
      DADD    D520 K5000 D8360
      DMOV    K0 D54
      SET     M323  ; 左臂上下速度设定
15605 LD      M187  ; 不在原点
      OUT     T56 K1  ; 不在原点
      ANDP    T56  ; 不在原点
      SET     M237  ; 左臂上下马达运行
15612 LD      M187  ; 不在原点
      AND     M622  ; X22-左臂上下原点
      OUT     T57 K2  ; 在原点
      AND     T57  ; 在原点
      RST     M187  ; 不在原点
      SET     M186  ; 在原点
15620 LDP     M186  ; 在原点
      DMOV    K0 D54
      DMOV    K-5000 D8360
      DMOV    K300 D50
15649 LD      M186  ; 在原点
      OUT     T58 K1  ; 在原点2
      ANDP    T58  ; 在原点2
      SET     M237  ; 左臂上下马达运行
      SET     M323  ; 左臂上下速度设定
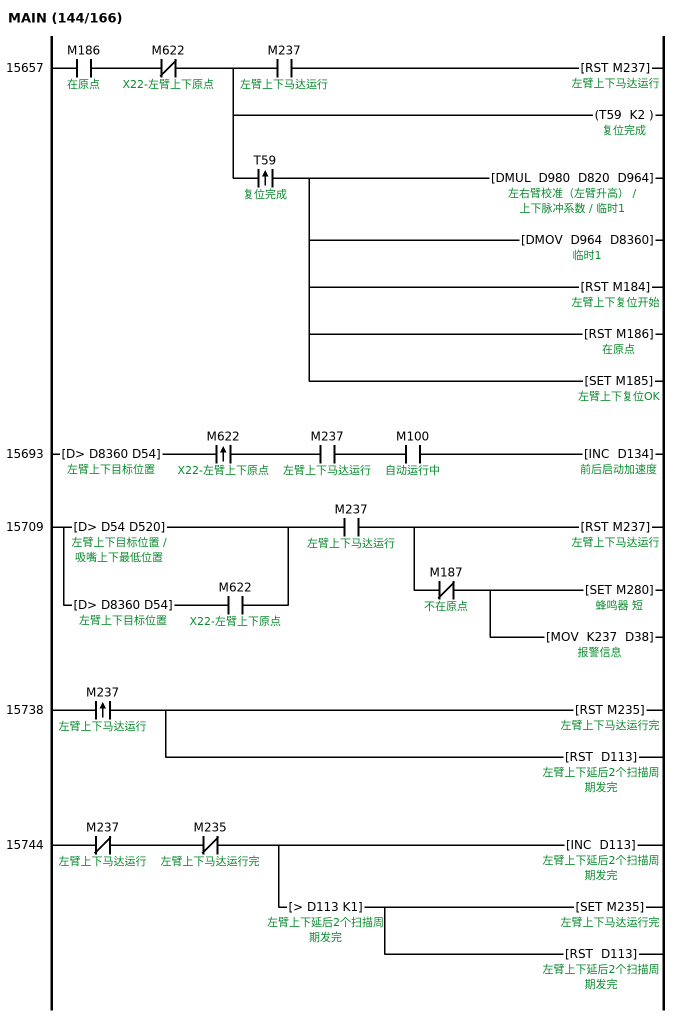
15657 LD      M186  ; 在原点
      ANI     M622  ; X22-左臂上下原点
      MPS
      AND     M237  ; 左臂上下马达运行
      RST     M237  ; 左臂上下马达运行
      MPP
      OUT     T59 K2  ; 复位完成
      ANDP    T59  ; 复位完成
      DMUL    D980 D820 D964
      DMOV    D964 D8360
      RST     M184  ; 左臂上下复位开始
      RST     M186  ; 在原点
      SET     M185  ; 左臂上下复位OK
15693 LDD>    D8360 D54  ; 左臂上下目标位置
      ANDP    M622  ; X22-左臂上下原点
      AND     M237  ; 左臂上下马达运行
      AND     M100  ; 自动运行中
      INC     D134  ; 前后启动加速度
15709 LDD>    D54 D520  ; 左臂上下目标位置 / 吸嘴上下最低位置
      LDD>    D8360 D54  ; 左臂上下目标位置
      AND     M622  ; X22-左臂上下原点
      ORB
      AND     M237  ; 左臂上下马达运行
      RST     M237  ; 左臂上下马达运行
      ANI     M187  ; 不在原点
      SET     M280  ; 蜂鸣器 短
      MOV     K237 D38
15738 LDP     M237  ; 左臂上下马达运行
      RST     M235  ; 左臂上下马达运行完
      RST     D113  ; 左臂上下延后2个扫描周期发完
15744 LDI     M237  ; 左臂上下马达运行
      ANI     M235  ; 左臂上下马达运行完
      INC     D113
      AND>    D113 K1  ; 左臂上下延后2个扫描周期发完
      SET     M235  ; 左臂上下马达运行完
      RST     D113  ; 左臂上下延后2个扫描周期发完
